{attribute 'estimated-stack-usage' := '8192'}
// Computes the number of bytes that would be needed to encode an
// embedded message field, including the tag.
FUNCTION F_ComputeMessageSize : UDINT
VAR_INPUT
    iMessage : I_Message;
END_VAR
VAR
	nSize	: UDINT;
    aBuffer : T_ProtobufRawBuffer;
    hr : HRESULT;
END_VAR


IF iMessage = NULL THEN
	RETURN;
END_IF

hr := iMessage.Writer.WriteTo(aBuffer);
IF FAILED(hr) THEN
    RETURN;
END_IF

nSize := iMessage.Writer.nBytesWritten;
F_ComputeMessageSize := F_ComputeLengthSize(nSize) + nSize;

END_FUNCTION

(* stored: Version 1.1.0.1
   POU F_ComputeMessageSize: Id {ee9eebb3-63b9-48a3-8f47-ea53b3104af8}, SpecialFunc None *)
